// TIA Portal V20 export
ORGANIZATION_BLOCK "Startup"   // OB1025, LAD, Startup
TITLE = "Complete Restart"
// stored: AutoNumber false, IsIECCheckEnabled true, Namespace Unit1.Em4, SetENOAutomatically true
   VAR_INPUT
      LostRetentive : Bool;   // True if retentive data are lost
      LostRTC : Bool;   // True if date and time are lost
   END_VAR
BEGIN

REGION Network 1 (SCL): Build the Absolut Reference Designator
   // Set the Absoult Reference Designator in the Config DB
   IF LEN(IN := "Unit1.Em4.Config".em.referenceDesignator.parent) <> 0 THEN
       "Unit1.Em4.Config".em.referenceDesignator.combined := CONCAT_WSTRING(IN1 := "Unit1.Em4.Config".em.referenceDesignator.parent, IN2 := WSTRING#'.', IN3 := "Unit1.Em4.Config".em.referenceDesignator.relative);
   ELSE
       "Unit1.Em4.Config".em.referenceDesignator.combined := "Unit1.Em4.Config".em.referenceDesignator.relative;
   END_IF;
END_REGION

REGION Network 2 (SCL): Assign axes data
   // This is an example how to assign axes to DB_ANY in DB Config. If you have axes, assign them here. The Config.axis[] variables will be handed over to the control modules. That enables a flexible programming.
   // Assign axes
   "Unit1.MotionNodes".PLCToMotion.TechnologyObject.Axis.Compensator := "Unit1.Em4.Config".axis[1] := "BA010AZCRDR3_CompensatorAxisZ";
   "Unit1.MotionNodes".PLCToMotion.TechnologyObject.Axis.FeedingRoller := "Unit1.Em4.Config".axis[2] := "BA010AZCRDR4_FeedingRollAxisB";
   "Unit1.MotionNodes".PLCToMotion.TechnologyObject.Axis.Cutter := "Unit1.Em4.Config".axis[3] := "BA010AZCRDR5_ElectordCutterAxisZ";
   "Unit1.Em4.Config".axis[4] := "BA010AZCRDR6_PositionMovingAxisX";

   // Cam
   "Unit1.MotionNodes".PLCToMotion.TechnologyObject.Cam.CompensatorCam1:="Unit1.Em4.Config".cam[1] := "BA010AZCRDR3_CompensatorAxisZCamMain_1";
   "Unit1.MotionNodes".PLCToMotion.TechnologyObject.Cam.CompensatorCam2:="Unit1.Em4.Config".cam[2] := "BA010AZCRDR3_CompensatorAxisZCamMain_2";
   "Unit1.MotionNodes".PLCToMotion.TechnologyObject.Cam.FeedingRollerCam1 := "Unit1.Em4.Config".cam[3] := "BA010AZCRDR4_FeedingRollAxisBCamMain_1";
   "Unit1.MotionNodes".PLCToMotion.TechnologyObject.Cam.FeedingRollerCam2 := "Unit1.Em4.Config".cam[4] := "BA010AZCRDR4_FeedingRollAxisBCamMain_2";
   "Unit1.MotionNodes".PLCToMotion.TechnologyObject.Cam.CutterCam := "Unit1.Em4.Config".cam[5] := "BA010AZCRDR5_ElectordCutterAxisZCamMain";

   // OutputCam
   //Config.OutputCam[1] :=
   "Unit1.Em4.Config".OutputCam[2] := "OutputCam_FeedingRollAxisB";
   "Unit1.Em4.Config".OutputCam[3] := "OutputCam_ElectordCutterAxisZ";
   //Config.OutputCam[4] :=

   // MeasuringInput
   "Unit1.MotionNodes".PLCToMotion.TechnologyObject.MeasureInput.Tab := "Unit1.Em4.Config".MeasuringInput[1] := "MeasuringInput_FeedingRollAxisB_Tab";
   "Unit1.MotionNodes".PLCToMotion.TechnologyObject.MeasureInput.Tape := "Unit1.Em4.Config".MeasuringInput[2] := "MeasuringInput_FeedingRollAxisB_Tape";
   //Config.MeasuringInput[3] := 
   //Config.MeasuringInput[4] :=

   // HW_SubModule
   "Unit1.Em4.Config".moduleAccessPoint[1] := "BA010AZCRCU1~BA010AZCRCU1_X150~BA010AZCRDR3_ModuleAccessPoint";
   "Unit1.Em4.Config".moduleAccessPoint[2] := "BA010AZCRCU1~BA010AZCRCU1_X150~BA010AZCRDR4_ModuleAccessPoint";
   "Unit1.Em4.Config".moduleAccessPoint[3] := "BA010AZCRCU2~BA010AZARCU2_X150~BA010AZCRDR5_ModuleAccessPoint";
   "Unit1.Em4.Config".moduleAccessPoint[4] := "BA010AZCRCU2~BA010AZARCU2_X150~BA010AZCRDR6_ModuleAccessPoint";

   // FB Enable
   "Unit1.Em4.HmiInterface".cmCompensatorAxisZ.commands.enable := TRUE;
   "Unit1.Em4.HmiInterface".cmFeedingRollAxisB.commands.enable := TRUE;
   "Unit1.Em4.HmiInterface".cmElectrodeCutterAxisZ.commands.enable := TRUE;
   "Unit1.Em4.HmiInterface".cmPositionMovingAxisX.commands.enableMasterControl := TRUE;

   // Assign configuration Homing
   "Unit1.Em4.ControlNodes".cmCompensatorAxisZ.commandConfiguration.homing.mode := "Unit1.Em4.HmiInterface".cmCompensatorAxisZ.commandConfiguration.homing.mode := 3;
   "Unit1.Em4.ControlNodes".cmElectrodeCutterAxisZ.commandConfiguration.homing.mode := "Unit1.Em4.HmiInterface".cmElectrodeCutterAxisZ.commandConfiguration.homing.mode := 3;
   "Unit1.Em4.ControlNodes".cmPositionMovingAxisX.commandConfiguration.homing.mode := "Unit1.Em4.HmiInterface".cmPositionMovingAxisX.commandConfiguration.homing.mode := 3;
END_REGION

REGION Network 3 (SCL): CM Config
   // Compensator Axis Z
   "Unit1.Em4.Config".cmCompensatorAxisZ.referenceDesignator := WSTRING#'Compensator Axis Z';
   "Unit1.Em4.Config".cmCompensatorAxisZ.disableAlarms := FALSE;
   "Unit1.Em4.Config".cmCompensatorAxisZ.masterControlPopUp := TRUE;


   // Electrode Cutter Axis Z
   "Unit1.Em4.Config".cmElectrodeCutterAxisZ.referenceDesignator := WSTRING#'Electrode Cutter Axis Z';
   "Unit1.Em4.Config".cmElectrodeCutterAxisZ.disableAlarms := FALSE;
   "Unit1.Em4.Config".cmElectrodeCutterAxisZ.masterControlPopUp := TRUE;


   // Feeding Roll Axis B
   "Unit1.Em4.Config".cmFeedingRollAxisB.referenceDesignator := WSTRING#'Feeding Roll Axis B';
   "Unit1.Em4.Config".cmFeedingRollAxisB.disableAlarms := FALSE;
   "Unit1.Em4.Config".cmFeedingRollAxisB.masterControlPopUp := TRUE;


   // Position Moving Axis X
   "Unit1.Em4.Config".cmPositionMovingAxisX.referenceDesignator := WSTRING#'Position Moving Axis X';


   // Feeder Cylinder
   "Unit1.Em4.Config".cmFeederCylinderUpDown.referenceDesignator := WSTRING#'Feeder Cylinder';
   "Unit1.Em4.Config".cmFeederCylinderUpDown.monitoringLeavingFeedback := T#5s;
   "Unit1.Em4.Config".cmFeederCylinderUpDown.monitoringReachingFeedback := T#5s;
   "Unit1.Em4.Config".cmFeederCylinderUpDown.monitoringDiscrepancy := T#0ms;
   "Unit1.Em4.Config".cmFeederCylinderUpDown.setOutputHomeContinuously := TRUE;
   "Unit1.Em4.Config".cmFeederCylinderUpDown.setOutputWorkContinuously := TRUE;
   "Unit1.Em4.Config".cmFeederCylinderUpDown.disableHomeCommand := FALSE;
   "Unit1.Em4.Config".cmFeederCylinderUpDown.disableFeedbackHomePos := FALSE;
   "Unit1.Em4.Config".cmFeederCylinderUpDown.disableFeedbackWorkPos := FALSE;
   "Unit1.Em4.Config".cmFeederCylinderUpDown.disableAlarms := FALSE;
   "Unit1.Em4.Config".cmFeederCylinderUpDown.resetOutputsOnError := FALSE;
   "Unit1.Em4.Config".cmFeederCylinderUpDown.allwaysWaitOnReachingTime := FALSE;


   // Compensator Safety Pin Idle Position
   "Unit1.Em4.Config".cmCompensatorSafetyPinIdlePosition.referenceDesignator := WSTRING#'DigitalSignal';
   "Unit1.Em4.Config".cmCompensatorSafetyPinIdlePosition.onDelay := T#0ms;
   "Unit1.Em4.Config".cmCompensatorSafetyPinIdlePosition.offDelay := T#0ms;
   "Unit1.Em4.Config".cmCompensatorSafetyPinIdlePosition.default := FALSE;
   "Unit1.Em4.Config".cmCompensatorSafetyPinIdlePosition.invertProcessValue := FALSE;
   "Unit1.Em4.Config".cmCompensatorSafetyPinIdlePosition.disableAlarms := FALSE;


   // Cutter Epc
   "Unit1.Em4.Config".cmCutterEpcAnalogInput.referenceDesignator := WSTRING#'Load Cell AnalogInput';
   "Unit1.Em4.Config".cmCutterEpcAnalogInput.physicalUnit := 'mm';
   "Unit1.Em4.Config".cmCutterEpcAnalogInput.isUnipolarSignal := TRUE;
   "Unit1.Em4.Config".cmCutterEpcAnalogInput.default := 0;
   "Unit1.Em4.Config".cmCutterEpcAnalogInput.limitHigh2 := 100;
   "Unit1.Em4.Config".cmCutterEpcAnalogInput.limitHigh1 := 90;
   "Unit1.Em4.Config".cmCutterEpcAnalogInput.limitLow1 := -90;
   "Unit1.Em4.Config".cmCutterEpcAnalogInput.limitLow2 := -100;
   "Unit1.Em4.Config".cmCutterEpcAnalogInput.processValueMax := 100;
   "Unit1.Em4.Config".cmCutterEpcAnalogInput.processValueMin := -100;
   "Unit1.Em4.Config".cmCutterEpcAnalogInput.scaleAnalogUppPoint := 27648;
   "Unit1.Em4.Config".cmCutterEpcAnalogInput.scaleAnalogLowPoint := 0;
   "Unit1.Em4.Config".cmCutterEpcAnalogInput.scaleProcessUppPoint := 100;
   "Unit1.Em4.Config".cmCutterEpcAnalogInput.scaleProcessLowPoint := -100;
   "Unit1.Em4.Config".cmCutterEpcAnalogInput.disableAlarms := FALSE;


   // Alarm Count referenceDesignator
   "Unit1.Em4.HmiInterface".cutterLifeCount.referenceDesignator := WSTRING#'Cutter Life Count';
   "Unit1.Em4.HmiInterface".tabSensorNotDetectedCount.referenceDesignator := WSTRING#'Tab Sensor Not Detected Count';


   // Softcam
   //HmiInterface.cm.softcam.positionMoving.UnitName := WSTRING#'mm';
END_REGION
END_ORGANIZATION_BLOCK
